// Mitsubishi GX Works2 project: 신호등   PLC: Q02/Q02H

PROGRAM MAIN
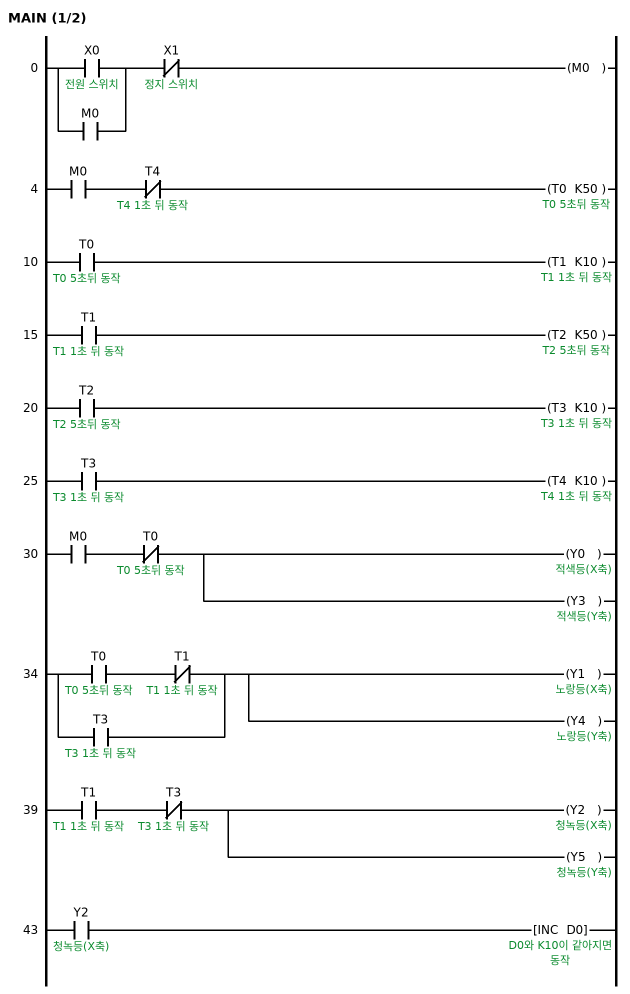
0     LD      X0  ; 전원 스위치
      OR      M0
      ANI     X1  ; 정지 스위치
      OUT     M0
4     LD      M0
      ANI     T4  ; T4 1초 뒤 동작
      OUT     T0 K50  ; T0 5초뒤 동작
10    LD      T0  ; T0 5초뒤 동작
      OUT     T1 K10  ; T1 1초 뒤 동작
15    LD      T1  ; T1 1초 뒤 동작
      OUT     T2 K50  ; T2 5초뒤 동작
20    LD      T2  ; T2 5초뒤 동작
      OUT     T3 K10  ; T3 1초 뒤 동작
25    LD      T3  ; T3 1초 뒤 동작
      OUT     T4 K10  ; T4 1초 뒤 동작
30    LD      M0
      ANI     T0  ; T0 5초뒤 동작
      OUT     Y0  ; 적색등(X축)
      OUT     Y3  ; 적색등(Y축)
34    LD      T0  ; T0 5초뒤 동작
      ANI     T1  ; T1 1초 뒤 동작
      OR      T3  ; T3 1초 뒤 동작
      OUT     Y1  ; 노랑등(X축)
      OUT     Y4  ; 노랑등(Y축)
39    LD      T1  ; T1 1초 뒤 동작
      ANI     T3  ; T3 1초 뒤 동작
      OUT     Y2  ; 청녹등(X축)
      OUT     Y5  ; 청녹등(Y축)
43    LD      Y2  ; 청녹등(X축)
      INC     D0  ; D0와 K10이 같아지면 동작
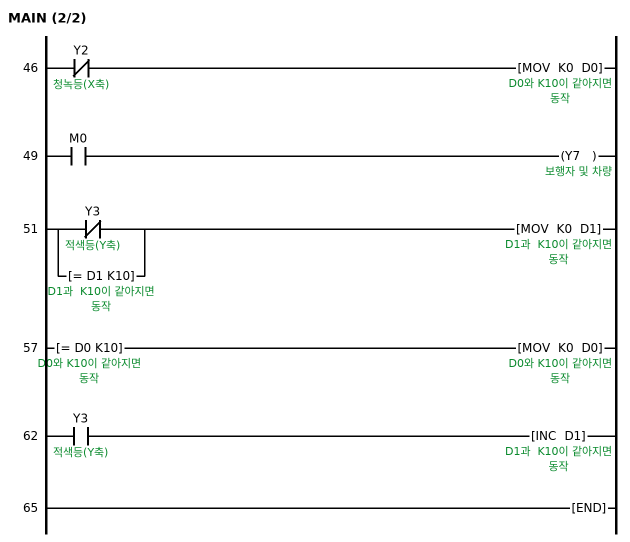
46    LDI     Y2  ; 청녹등(X축)
      MOV     K0 D0
49    LD      M0
      OUT     Y7  ; 보행자 및 차량
51    LDI     Y3  ; 적색등(Y축)
      OR=     D1 K10  ; D1과  K10이 같아지면 동작
      MOV     K0 D1
57    LD=     D0 K10  ; D0와 K10이 같아지면 동작
      MOV     K0 D0
62    LD      Y3  ; 적색등(Y축)
      INC     D1
65    END
END_PROGRAM
